FUNCTION_BLOCK number
VAR
	number 		at %I* : int;
END_VAR

END_FUNCTION_BLOCK

(* stored: Version 1.1.0.1
   POU number: Id {35d5f773-f920-47e3-8c55-ef80baae71ee}, SpecialFunc None *)
